FUNCTION_BLOCK FB_MGMT
VAR_INPUT
	Freigabe_auto			: BOOL;
	Freigabe_Deakt_auto		: BOOL;
	Betrieb_Anford_auto		: BOOL;
	Regelung_Modus_auto		: SINT;
	Regelung_Sollw_auto		: REAL;
END_VAR
VAR_OUTPUT
END_VAR
VAR
	Netze_MGMT		    	: FB_MGMT_ThNTZ;
	Betonspeicher			: FB_MGMT_BSp;

	{attribute 'OPC.UA.DA' := '1'}Steuerung				: ST_FB_MGMT_Steuerung;		
	{attribute 'OPC.UA.DA' := '1'}Stellwert				: ST_FB_MGMT_Stellwert;		
	{attribute 'OPC.UA.DA' := '1'}Zustand					: ST_FB_MGMT_Zustand;	
	{attribute 'OPC.UA.DA' := '1'}Parameter				: ST_FB_MGMT_Parameter;		

    Zustandscheck			: FB_MGMT_Zustandscheck;
	Logik					: FB_MGMT_Logik;
	Ablaufsteuerung			: FB_MGMT_Ablaufsteuerung;
	Sollwertscheck			: FB_MGMT_Sollwertscheck;
	Regelung				: FB_MGMT_Regelung;
	Zuweisungen				: FB_Zuweisungen;

END_VAR

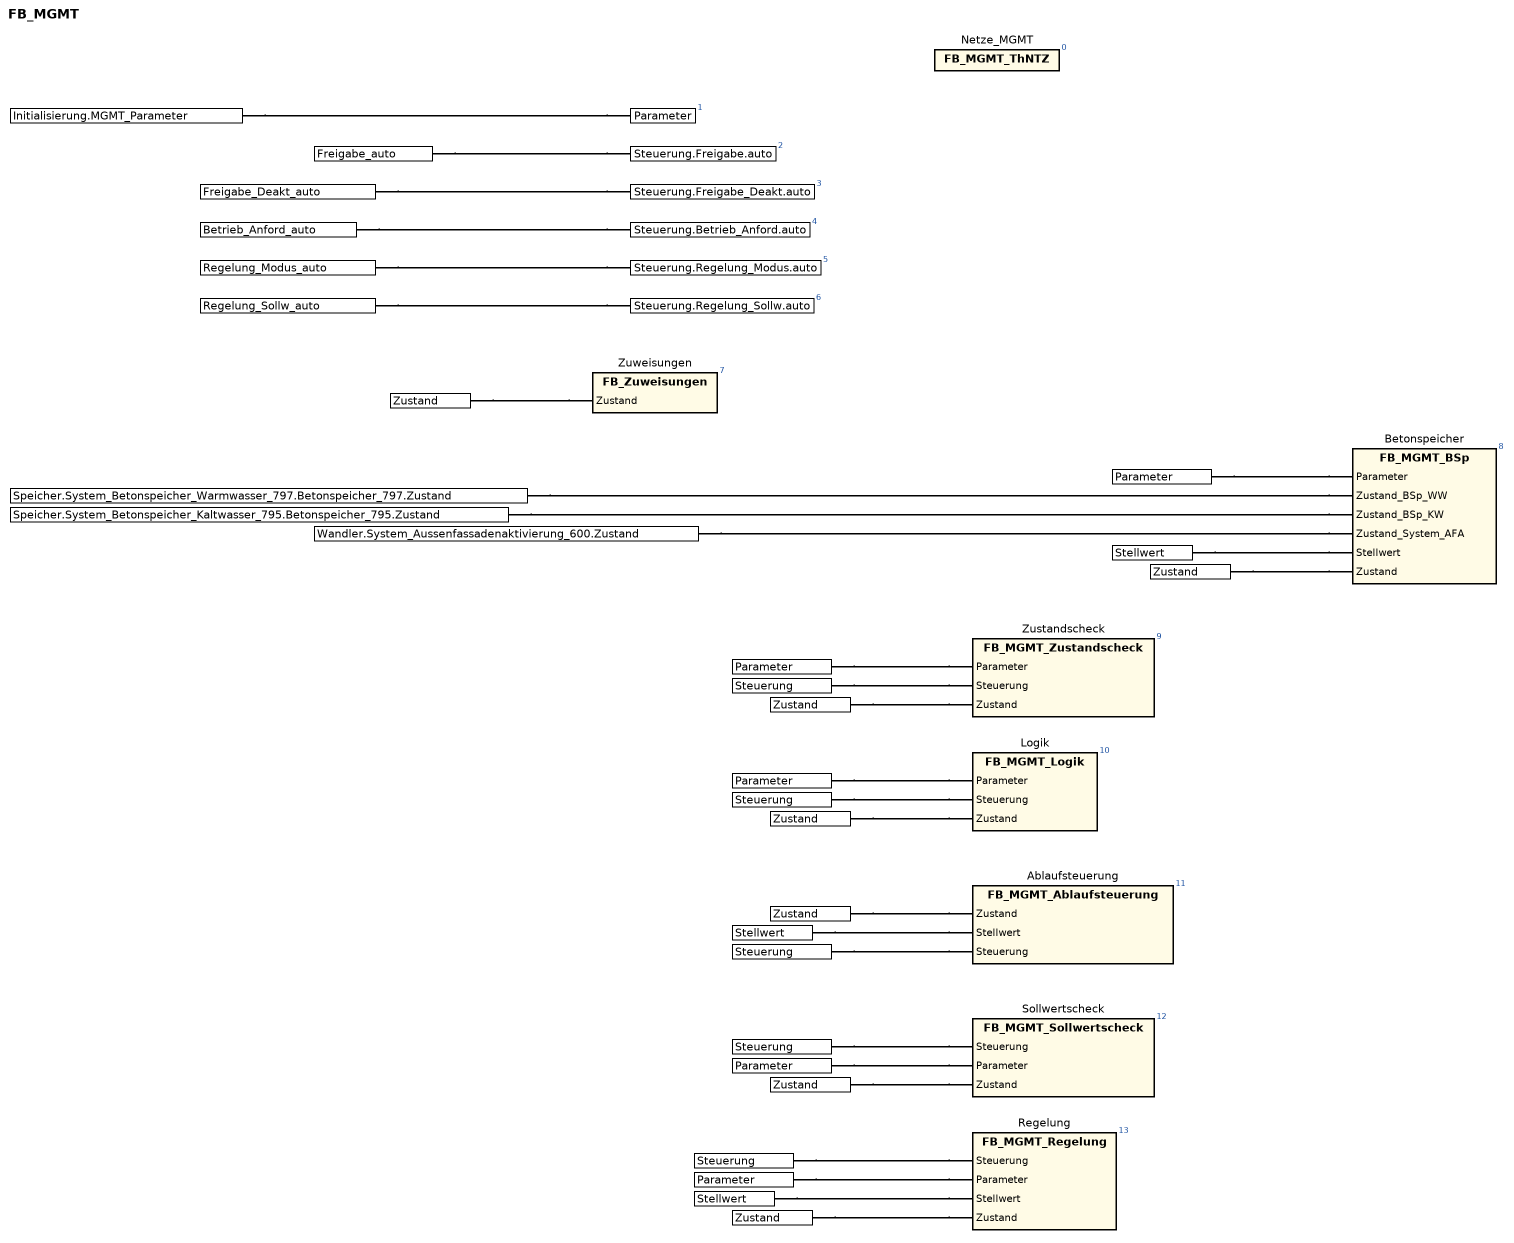
Netze_MGMT(); // FB_MGMT_ThNTZ
Parameter := Initialisierung.MGMT_Parameter;
Steuerung.Freigabe.auto := Freigabe_auto;
Steuerung.Freigabe_Deakt.auto := Freigabe_Deakt_auto;
Steuerung.Betrieb_Anford.auto := Betrieb_Anford_auto;
Steuerung.Regelung_Modus.auto := Regelung_Modus_auto;
Steuerung.Regelung_Sollw.auto := Regelung_Sollw_auto;
Zuweisungen(Zustand := Zustand); // FB_Zuweisungen
Betonspeicher(
    Parameter := Parameter,
    Zustand_BSp_WW := Speicher.System_Betonspeicher_Warmwasser_797.Betonspeicher_797.Zustand,
    Zustand_BSp_KW := Speicher.System_Betonspeicher_Kaltwasser_795.Betonspeicher_795.Zustand,
    Zustand_System_AFA := Wandler.System_Aussenfassadenaktivierung_600.Zustand,
    Stellwert := Stellwert,
    Zustand := Zustand); // FB_MGMT_BSp
Zustandscheck(Parameter := Parameter, Steuerung := Steuerung, Zustand := Zustand); // FB_MGMT_Zustandscheck
Logik(Parameter := Parameter, Steuerung := Steuerung, Zustand := Zustand); // FB_MGMT_Logik
Ablaufsteuerung(Zustand := Zustand, Stellwert := Stellwert, Steuerung := Steuerung); // FB_MGMT_Ablaufsteuerung
Sollwertscheck(Steuerung := Steuerung, Parameter := Parameter, Zustand := Zustand); // FB_MGMT_Sollwertscheck
Regelung(Steuerung := Steuerung, Parameter := Parameter, Stellwert := Stellwert, Zustand := Zustand); // FB_MGMT_Regelung

END_FUNCTION_BLOCK

(* stored: Version 1.1.0.1, ProductVersion 3.1.4024.9
   POU FB_MGMT: Id {683854d9-e7d5-4abb-b208-33dbae93ac7f}, SpecialFunc None *)
